// Mitsubishi GX Works2 project: 20150630   PLC: Q03UDV

PROGRAM P1
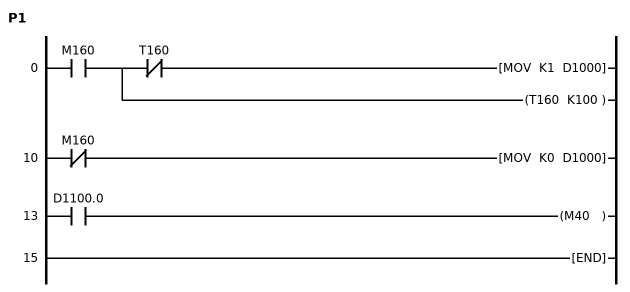
0     LD      M160
      MPS
      ANI     T160
      MOV     K1 D1000
      MPP
      OUT     T160 K100
10    LDI     M160
      MOV     K0 D1000
13    LD      D1100.0
      OUT     M40
15    END
END_PROGRAM

PROGRAM P2
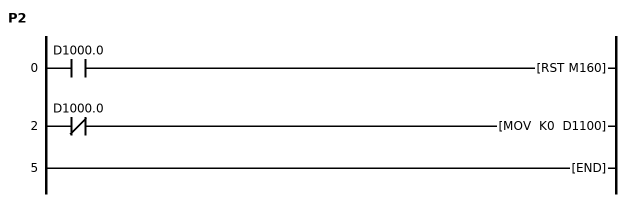
0     LD      D1000.0
      RST     M160
2     LDI     D1000.0
      MOV     K0 D1100
5     END
END_PROGRAM
